{attribute 'qualified_only'}
{attribute 'strict'}
TYPE ParallelStates :
(
	Idle := 0, Startup, Standalone, Slave, Master
);
END_TYPE

(* stored: Version 1.1.0.1, ProductVersion 3.1.4024.6
   DUT ParallelStates: Id {1bad3a29-4217-462d-a5a2-1342394668f5} *)
